FUNCTION_BLOCK MultiIDischarge (* Composite Function Block Type *)
  (* Standard: 61499-2 *)
  (* Version 0.0, 8/28/2026, Schneider Electric, template *)
  PACKAGE SE.Nereda;
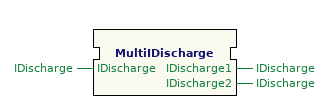
  SOCKETS
    IDischarge : IDischarge;
  END_SOCKETS
  PLUGS
    IDischarge1 : IDischarge;
    IDischarge2 : IDischarge;
  END_PLUGS
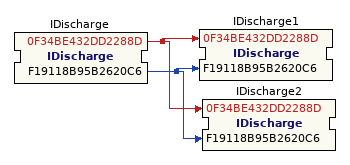
  EVENT_CONNECTIONS
    IDischarge.0F34BE432DD2288D TO IDischarge1.0F34BE432DD2288D;
    IDischarge.0F34BE432DD2288D TO IDischarge2.0F34BE432DD2288D;
  END_CONNECTIONS
  DATA_CONNECTIONS
    IDischarge.F19118B95B2620C6 TO IDischarge1.F19118B95B2620C6;
    IDischarge.F19118B95B2620C6 TO IDischarge2.F19118B95B2620C6;
  END_CONNECTIONS
END_FUNCTION_BLOCK
